Fanuc KAREL source: kt00979.KL

-- PROVISIONAL review KL for V1013-1; original PC SHA256 83049579d2c099fd4a08814c530a8219e8577a6b8b9fdcaaf6e3b328bcee5008
-- Incomplete behavior may be omitted. Consult companion uncertainty JSON. Do not deploy.
PROGRAM KT00979
%NOLOCKGROUP
VAR
  I1 : INTEGER
  I2 : INTEGER
-- UNRESOLVED_DECL CFG type=00001c
-- UNRESOLVED_DECL OUT type=000101
BEGIN
  -- UNRESOLVED_PC offsets 5-16; opcodes 2E,23
  -- UNRESOLVED_PC offsets 21-32; opcodes 2E,23
  -- UNRESOLVED_PC offsets 37-48; opcodes 2E,23
  -- UNRESOLVED_PC offsets 53-64; opcodes 2E,23
  -- UNRESOLVED_PC offsets 69-79; opcodes 9D,22,A5
  -- UNRESOLVED_PC offsets 84-153; opcodes 27,27,21,64,27,21,64,27,21,64,27,21,64,27,21,64,27,21,64,22,76,7E,4A
  -- UNRESOLVED_PC offsets 158-162; opcodes 7F
END KT00979
